FUNCTION_BLOCK FB_Control_Estacion
VAR_INPUT
	Start_Button : BOOL;
	Stop_Button : BOOL;
	Reset_Button : BOOL;
	Safety_Door : BOOL;
	
END_VAR
VAR_IN_OUT
	Estado             : INT;
END_VAR
VAR_OUTPUT
	Control 		   : BOOL;
	Start_Button_Light : BOOL;
	Stop_Button_Light  : BOOL;
	Reset_Button_Light : BOOL;
	Stack_Light_Green  : BOOL;	 
	Stack_Light_Red    : BOOL;	
	Stack_Light_Yellow : BOOL;
	
END_VAR
VAR	
END_VAR

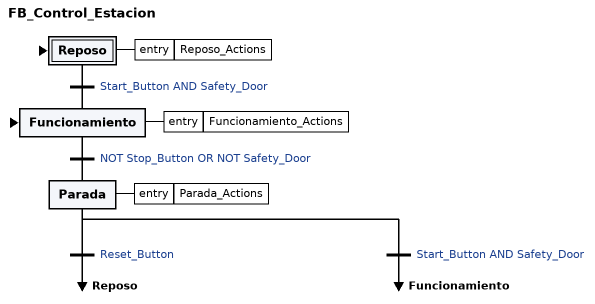
INITIAL_STEP Reposo:
    Reposo_Actions(P1);  // entry action
END_STEP
TRANSITION FROM Reposo TO Funcionamiento
    := Start_Button AND Safety_Door;
END_TRANSITION
STEP Funcionamiento:
    Funcionamiento_Actions(P1);  // entry action
END_STEP
TRANSITION FROM Funcionamiento TO Parada
    := NOT Stop_Button OR NOT Safety_Door;
END_TRANSITION
STEP Parada:
    Parada_Actions(P1);  // entry action
END_STEP
TRANSITION FROM Parada TO Reposo
    := Reset_Button;
END_TRANSITION
TRANSITION FROM Parada TO Funcionamiento
    := Start_Button AND Safety_Door;
END_TRANSITION

ACTION Funcionamiento_Actions:
Control := TRUE; // Se indica que la estación puede funcionar
// Se indica mediante una luz que el siguiente botón a pulsar sería el de Stop
Start_Button_Light := FALSE;
Stop_Button_Light := TRUE;
Reset_Button_Light := FALSE;
//Semáforo indicando estación en funcionamiento
Stack_Light_Green := TRUE; 
Stack_Light_Red := FALSE;	
Stack_Light_Yellow := FALSE;
END_ACTION

ACTION Parada_Actions:
Control := FALSE; // Se indica que la estación no puede funcionar
// Se indica mediante una luz que el siguiente botón a pulsar sería el de Stop o el reset dependiendo de la acción deseada
Stop_Button_Light := FALSE;
Start_Button_Light := TRUE;
Reset_Button_Light := TRUE;
//Semáforo indicando que se ha solicitado la parada de la estación
Stack_Light_Green := FALSE;
Stack_Light_Red := FALSE;	
Stack_Light_Yellow := TRUE;
END_ACTION

ACTION Reposo_Actions:
Control := FALSE; // Se indica que la planta no puede funcionar
// Se indica mediante una luz que el siguiente botón a pulsar sería el de Start
Start_Button_Light := TRUE;
Stop_Button_Light := FALSE;
Reset_Button_Light := FALSE;
Estado := 0;
//Semáforo indicando estación parada
Stack_Light_Green := FALSE;	 
Stack_Light_Red := TRUE;	
Stack_Light_Yellow := FALSE;
END_ACTION

END_FUNCTION_BLOCK

(* stored: Version 1.1.0.1, ProductVersion 3.1.4024.12
   POU FB_Control_Estacion: Id {52f3885c-340e-46e1-b2b5-b332c43ff229}, SpecialFunc None
   Action Funcionamiento_Actions: Id {2d478830-46ef-4e81-ad66-c9651a3719d9}
   Action Parada_Actions: Id {2d444389-3a8b-4e75-92c2-8c82de2620f2}
   Action Reposo_Actions: Id {558b7fda-f947-4b5b-97d6-fe187eecd04a} *)
